TYPE ST_St020_IO_OUT :
STRUCT
	bOvenFan :BOOL;
END_STRUCT
END_TYPE

(* stored: Version 1.1.0.1
   DUT ST_St020_IO_OUT: Id {f5be0bc9-568b-49ad-994f-e78c80690e21} *)
